# EPICS substitutions: splineApp/Db/k_to_gap.substitutions
file spline.template

{
  pattern{ DEV, LOCA, UNIT, FILENAME }
         { UND, B81, MC, pid_fit_k.data}

}
